FUNCTION_BLOCK StartStop (* Basic Function Block Type *)
  (* Standard: 61499-2 *)
  (* Version 0.0, 18/05/2022, Admin, Schneider Electric, Template *)
  PACKAGE Main;
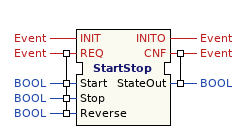
  EVENT_INPUT
    INIT; (* Initialization Request *)
    REQ WITH Start, Stop, Reverse; (* Normal Execution Request *)
  END_EVENT
  EVENT_OUTPUT
    INITO; (* Initialization Confirm *)
    CNF WITH StateOut; (* Execution Confirmation *)
  END_EVENT
  VAR_INPUT
    Start : BOOL; (* Input event qualifier *)
    Stop : BOOL;
    Reverse : BOOL;
  END_VAR
  VAR_OUTPUT
    StateOut : BOOL; (* Output event qualifier *)
  END_VAR
  VAR
    InternalState : BOOL;
  END_VAR
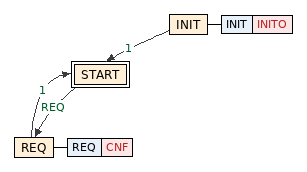
  EC_STATES
    START; (* Initial State *)
    INIT : INIT -> INITO; (* Initialization *)
    REQ : REQ -> CNF; (* Normal execution *)
  END_STATES
  EC_TRANSITIONS
    INIT TO START := 1;
    START TO REQ := REQ;
    REQ TO START := 1;
  END_TRANSITIONS
  ALGORITHM INIT IN ST: (* Initialization algorithm *)
;
  END_ALGORITHM
  ALGORITHM REQ IN ST: (* Normally executed algorithm *)
;

InternalState := AND(XOR(OR(Start, InternalState), Reverse), NOT(Stop));

StateOut := InternalState;
  END_ALGORITHM
END_FUNCTION_BLOCK
